// Mitsubishi GX Works2 project: b03   PLC: Q02/Q02H

PROGRAM MAIN
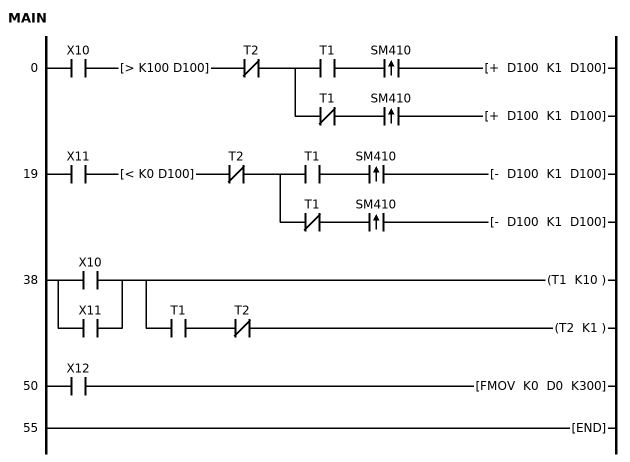
0     LD      X10
      AND>    K100 D100
      ANI     T2
      MPS
      AND     T1
      ANDP    SM410
      +       D100 K1 D100
      MPP
      ANI     T1
      ANDP    SM410
      +       D100 K1 D100
19    LD      X11
      AND<    K0 D100
      ANI     T2
      MPS
      AND     T1
      ANDP    SM410
      -       D100 K1 D100
      MPP
      ANI     T1
      ANDP    SM410
      -       D100 K1 D100
38    LD      X10
      OR      X11
      OUT     T1 K10
      AND     T1
      ANI     T2
      OUT     T2 K1
50    LD      X12
      FMOV    K0 D0 K300
55    END
END_PROGRAM
